PROGRAM MAIN
VAR
	INMODE : INMODE;
	
	CircularTablePosition1 : BOOL;
	CircularTablePosition2 : BOOL;
	CircularTablePosition3 : BOOL;
	PickupPointOccupied : BOOL; //NC gives back 1 when empty
	ManipulatorCircularEND : BOOL;
	ManipulatorFurnaceEND : BOOL;
	FurnaceIN : BOOL;
	FurnaceOUT : BOOL;
	FurnaceNotFULL : BOOL; //NC gives back 1 when empty
	CodeReader0 :  BOOL;
	CodeReader1 :  BOOL;
	StartButton : BOOL; //NO gives back 0 when not pressed
	SYSTEM_OK : BOOL;
	InConveyorOccupied : BOOL; //NO Gives back 0 when empty
	RobotIN_task_IN_Progress : BOOL;
	RobotOUT_task_IN_Progress : BOOL;
	
	CircTableRight : BOOL;
	CircTableLeft  : BOOL;
	PickupMotorGO : BOOL;
	SawMotor : BOOL;
	FurnaceGOin : BOOL;
	FurnaceGOout : BOOL;
	ManipulatorGOtoFurnace : BOOL;
	ManipulatorGOtoCircular : BOOL;
	FurnaceON : BOOL;
	ReaderTrigger : BOOL;
	ManipulatorVacuumON : BOOL; //monostabil
	ManipulatorZDOWN : BOOL; //monostabil!!!!!!
	FurnaceDoorUP :BOOL :=TRUE; //monostabil!!!!
 	RobotCOM0 : BOOL;
	RobotCOM1 : BOOL;
	CircularEJECT : BOOL; //monostabil!!!
	DelayTimer : TON;
	DelayAmount : TIME;
	DelayONtrigger : BOOL;
	FallTrig : F_TRIG;
	FallTrigCLK : BOOL;
	Pulse : Pulse;
	PulseSIGNAL : BOOL; 
	PulseTime : TIME;
	
	ScanCounter :INT := 0;
	FurnaceBurntime : TIME;
	
END_VAR

INMODE(); 
DelayTimer(IN:=DelayONtrigger,PT:=DelayAmount);
FallTrig(CLK:=FallTrigCLK);
Pulse(SIGNAL:=PulseSIGNAL,Pulse_time:=PulseTime);
CircularTablePosition1 := GIOL.In0;
CircularTablePosition2 := GIOL.In1;
CircularTablePosition3 := GIOL.In3;
PickupPointOccupied := GIOL.In2;
ManipulatorCircularEND := GIOL.In4;
ManipulatorFurnaceEND := GIOL.In7;
FurnaceIN := GIOL.In5;
FurnaceOUT := GIOL.In6;
FurnaceNotFULL := GIOL.In8;
CodeReader0 := GIOL.In9;
CodeReader1 := GIOL.In10;
StartButton := GIOL.In11;
SYSTEM_OK := GIOL.In12;
InConveyorOccupied := GIOL.In13;
RobotIN_task_IN_Progress := GIOL.In14;
RobotOUT_task_IN_Progress := GIOL.In15;

GIOL.Out0 := CircTableRight;
GIOL.Out1 := CircTableLeft;
GIOL.Out2 := PickupMotorGO;
GIOL.Out3 := SawMotor;
GIOL.Out4 := FurnaceGOin;
GIOL.Out5 := FurnaceGOout;
GIOL.Out6 := ManipulatorGOtoFurnace;
GIOL.Out7 := ManipulatorGOtoCircular;
GIOL.Out8 := FurnaceON;
GIOL.Out9 := ReaderTrigger;
GIOL.Out10 := ManipulatorVacuumON;
GIOL.Out11 := ManipulatorZDOWN;
GIOL.Out12 := FurnaceDoorUP;
GIOL.Out13 := RobotCOM0;
GIOL.Out14 := RobotCOM1;
GIOL.Out15 := CircularEJECT;

IF SYSTEM_OK THEN
CASE GIOL.CaseNum OF
	
	0:GIOL.TaskName:="Idle position, wait for start button";
		IF StartButton THEN
			GIOL.CaseNum:=10;
		END_IF
		
	10:GIOL.TaskName:="Check for workpiece on inconveyor";
		IF InConveyorOccupied AND FurnaceNotFULL THEN
			DelayAmount := T#1S;
			GIOL.CaseNum := 20;
		ELSE 
			GIOL.CaseNum:=0;
		END_IF
		
	20:GIOL.TaskName:="Wait for 1 sec";
		DelayONtrigger := TRUE;
		IF DelayTimer.Q THEN
			DelayONtrigger := FALSE;
			GIOL.CaseNum:=30;
		END_IF
		
	30:GIOL.TaskName:="Open furnace if in";
		IF FurnaceOUT THEN
			GIOL.CaseNum := 40;
		ELSE
			FurnaceGOout := TRUE;
			FurnaceGOin :=FALSE;
			DelayAmount := T#4S;
			GIOL.CaseNum := 35;
		END_IF
		
	35:GIOL.TaskName:="Open Furnace";
		DelayONtrigger := TRUE;
		IF DelayTimer.Q THEN
			GIOL.CaseNum := 40;
			DelayONtrigger := FALSE;
			FurnaceGOin := FALSE;
		END_IF
		
	40:GIOL.TaskName:="Give Robot load command";
		RobotCOM0 := 0;
		RobotCOM1 := 1;
		GIOL.CaseNum := 50;
		
	50:GIOL.TaskName:="Load workpiece into furnace";
		FallTrigCLK := RobotIN_task_IN_Progress;
		IF RobotIN_task_IN_Progress THEN
			RobotCOM0 := 0;
			RobotCOM1 := 0;
		END_IF
		IF FallTrig.Q THEN
			GIOL.CaseNum := 60;
		END_IF
		
	60:GIOL.TaskName:="Identify workpiece";
		IF NOT FurnaceNotFULL THEN
			ReaderTrigger := TRUE;
			PulseTime:=T#250MS;
			PulseSIGNAL:=TRUE;
			GIOL.CaseNum:=61;
		END_IF
	
	61:GIOL.TaskName:="Identify workpiece";
		IF NOT PulseSIGNAL THEN
			PulseTime:=T#2S;
			PulseSIGNAL:=TRUE;
			GIOL.CaseNum := 62;
			ReaderTrigger:=FALSE;
		END_IF
		
	62:GIOL.TaskName:="Identify workpiece";
		IF NOT PulseSIGNAL AND NOT CodeReader0 AND NOT CodeReader1 THEN
			ScanCounter := ScanCounter + 1;
			GIOL.CaseNum:=60;
			IF ScanCounter = 2 THEN
				GIOL.CaseNum:=0;
				ScanCounter:=0;
			END_IF
		END_IF
		
		IF NOT CodeReader0 AND CodeReader1 THEN
			FurnaceBurntime := T#5000MS;
			GIOL.CaseNum := 70;
		END_IF
		IF CodeReader0 AND NOT CodeReader1 THEN
			FurnaceBurntime := T#1500MS;
			GIOL.CaseNum := 70;
		END_IF
		IF CodeReader0 AND CodeReader1 THEN
			FurnaceBurntime := T#3000MS;
			GIOL.CaseNum := 70;
		END_IF
	
	70:GIOL.TaskName:="Pull workpiece into furnace";
		FurnaceGOin:=TRUE;
		FurnaceGOout:=FALSE;	
		GIOL.CaseNum:=71;
		ScanCounter:=0;
		
	71:GIOL.TaskName:="Pull workpiece into furnace";
		IF FurnaceIN THEN
			FurnaceGOin:=FALSE;
			FurnaceGOout:=FALSE;
			FurnaceDoorUP:=FALSE;
			DelayAmount:=T#1S;
			GIOL.CaseNum:=72;
		END_IF
	72:GIOL.TaskName:="Close furnace door";
		DelayONtrigger:=TRUE;
		IF DelayTimer.Q THEN
			DelayONtrigger:=FALSE;
			GIOL.CaseNum:=73;
			FurnaceON:=TRUE;
			DelayAmount:=FurnaceBurntime;
		END_IF
	73:GIOL.TaskName:="BURN!!!!";
		DelayONtrigger:=TRUE;
		IF DelayTimer.Q THEN
			DelayONtrigger:=FALSE;
			FurnaceON:=FALSE;
			FurnaceDoorUP:=TRUE;
			DelayAmount:=T#1S;
			GIOL.CaseNum:=80;
		END_IF
		
	80:GIOL.TaskName:="Open furnace door";
		DelayONtrigger:=TRUE;
		IF DelayTimer.Q THEN
			DelayONtrigger:=FALSE;
			FurnaceGOout:=TRUE;
			FurnaceGOin:=FALSE;
			GIOL.CaseNum:=90;
		END_IF
		
	90:GIOL.TaskName:="Send out workpiece";
		IF FurnaceOUT THEN
			ManipulatorGOtoFurnace:=TRUE;
			ManipulatorGOtoCircular:=FALSE;
			IF CircularTablePosition1 THEN
				GIOL.CaseNum:=100;
			ELSE
				GIOL.CaseNum:=91;
				CircTableLeft:=TRUE;
			END_IF			
		END_IF
		
	91:GIOL.TaskName:="Adjust circular table";
		IF CircularTablePosition1 THEN
			CircTableLeft := FALSE;
			GIOL.CaseNum  := 100;
		END_IF
		
	100:GIOL.TaskName:="Take workpiece to table";
		IF ManipulatorFurnaceEND THEN
			ManipulatorGOtoFurnace:=FALSE;
			ManipulatorGOtoCircular:=FALSE;
			ManipulatorZDOWN:=TRUE;
			ManipulatorVacuumON:=TRUE;
			DelayAmount:=T#1S;
			GIOL.CaseNum:=101;
		END_IF
		
	101:GIOL.TaskName:="Take workpiece to table";
		DelayONtrigger:=TRUE;
		IF DelayTimer.Q THEN
			DelayONtrigger:=FALSE;
			ManipulatorZDOWN:=FALSE;
			DelayAmount := T#500MS;
			GIOL.CaseNum:=102;
		END_IF
		
	102:GIOL.TaskName:="Take workpiece to table";
		DelayONtrigger:=TRUE;
		IF DelayTimer.Q THEN
			DelayONtrigger:=FALSE;
			ManipulatorGOtoCircular:=TRUE;
			GIOL.CaseNum:=103;
		END_IF
		
	103:GIOL.TaskName:="Take workpiece to table";
		IF ManipulatorCircularEND THEN
			ManipulatorZDOWN:=TRUE;
			DelayAmount:=T#500MS;
			GIOL.CaseNum:=104;
		END_IF
		
	104:GIOL.TaskName:="Take workpiece to table";
		DelayONtrigger:=TRUE;
		IF DelayTimer.Q THEN
			DelayONtrigger:=FALSE;
			ManipulatorVacuumON:=FALSE;
			ManipulatorZDOWN:=FALSE;
			DelayAmount:=T#500MS;
			GIOL.CaseNum:=105;
		END_IF
		
	105:GIOL.TaskName:="Wait for putdown";
		DelayONtrigger:=TRUE;
		IF DelayTimer.Q THEN
			CircTableRight:=TRUE;
			DelayONtrigger:=FALSE;
			GIOL.CaseNum:=110;
		END_IF
		
		
	110:GIOL.TaskName:="SAW Operation";
		IF CircularTablePosition3 THEN
			CircTableRight:=FALSE;
			SawMotor:=TRUE;
			DelayAmount:=T#2S;
			GIOL.CaseNum:=111;
		END_IF
	
	111:GIOL.TaskName:="SAW Operation";
		DelayONtrigger:=TRUE;
		IF DelayTimer.Q THEN
			DelayONtrigger:=FALSE;
			SawMotor:=FALSE;
			CircTableRight:=TRUE;
			GIOL.CaseNum:=120;
		END_IF
		
	120:GIOL.TaskName:="SAW Operation";
		IF CircularTablePosition2 THEN
			CircTableRight:=FALSE;
			DelayAmount:=T#500MS;
			GIOL.CaseNum:=130;
		END_IF
		
	130:GIOL.TaskName:="Eject workpiece from table";
		DelayONtrigger:=TRUE;
		IF DelayTimer.Q THEN
			DelayONtrigger:=FALSE;
			CircularEJECT:=TRUE;
			DelayAmount:=T#1000MS;
			GIOL.CaseNum:=131;
		END_IF
		
	131:GIOL.TaskName:="Eject workpiece from table";
		DelayONtrigger:=TRUE;
		IF DelayTimer.Q THEN
			DelayONtrigger:=FALSE;
			CircularEJECT:=FALSE;
			PickupMotorGO:=TRUE;
			CircTableLeft:=TRUE;
			GIOL.CaseNum:=140;
		END_IF
		
	140:GIOL.TaskName:="Take workpiece to pickup point";
		IF NOT PickupPointOccupied THEN
			PickupMotorGO:=FALSE;
		END_IF
		IF CircularTablePosition1 THEN 
			CircTableLeft:=FALSE;
			RobotCOM0:=1;
			RobotCOM1:=1;
			GIOL.CaseNum:=150;
		END_IF
			
	150:GIOL.TaskName:="Take workpiece to endpoint";
		FallTrigCLK :=  RobotOUT_task_IN_Progress;
		IF RobotOUT_task_IN_Progress THEN
			RobotCOM0 := 0;
			RobotCOM1 := 0;
		END_IF
		IF FallTrig.Q THEN
			GIOL.CaseNum := 160;
		END_IF
		
	160:GIOL.TaskName:="Finished task";
		GIOL.CaseNum:=10;
	
	ELSE
		GIOL.CaseNum:=0;
END_CASE
ELSE
	GIOL.CaseNum := 0;
	CircTableRight := 0;
	CircTableLeft := 0;
	PickupMotorGO := 0;
	SawMotor := 0;
	FurnaceGOin := 0;
	FurnaceGOout := 0;
	ManipulatorGOtoFurnace := 0;
	ManipulatorGOtoCircular := 0;
	RobotCOM0 := 0;
	RobotCOM1 :=0;
	FurnaceON := 0;
	ReaderTrigger := 0;
	ManipulatorVacuumON := 0;
	ManipulatorZDOWN := 0;
	CircularEJECT := 0;
END_IF
//some random change

END_PROGRAM

(* stored: Version 1.1.0.1, ProductVersion 3.1.4024.15
   POU MAIN: Id {55f2dad4-fae0-4be3-a7be-b728afd4fa9e}, SpecialFunc None *)
